TYPE ST_KNXnetIP_MessageOfAllGroupAddresses :
STRUCT
	aMessage		: ARRAY[0..31, 0..7, 0..255] OF ARRAY[1..255] OF BYTE;
END_STRUCT
END_TYPE

(* stored: Version 1.1.0.1
   DUT ST_KNXnetIP_MessageOfAllGroupAddresses: Id {2f68c5e4-4522-4881-ab06-1be81710f3d3} *)
